PROGRAM PRG_PID_CALL
VAR
	fbPlantControl : PlantAndCMs.FB_PlantControl_mode_2;
	Udt_FbPlantControl : PlantAndCMs.Udt_PlantControl_Mode_2;
	
	fbPlantModeSelector : PlantAndCMs.FB_ModeSelector;
	Udt_PlantModeSelector : PlantAndCMs.Udt_ModeSelector;
END_VAR

//aiSpare02c AT %I*: INT; //ch3 0-10v  Legacy range			(0-32767)
//measure 0-10v
//GVL.rAIInput1 := (INT_TO_REAL(IO.aiSpare02c)/(32767.0-0.0)) * 10.0;

//aiSpare02d AT %I*: INT; //ch4 0-20mA Extended range 		(0 -30518)
//measure 0-100%
//GVL.rAIInput2 := (INT_TO_REAL(IO.aiSpare02d)/(30518.0-0.0)) * 100.0;
fbPlantModeSelector(
	Ctrl_Data_ModeSelector := Udt_PlantModeSelector
	);

	
fbPlantControl(
	Start_In := PlantAndCMs.FIO.bStart,
	Stop_In := PlantAndCMs.FIO.bStop, 
	Reset_In := PlantAndCMs.FIO.bReset,
	
	
	Ctrl_Plant := Udt_FbPlantControl
	);

IF fbPlantControl.Startet_Out THEN
	//PRG_FB_CTRL_PID.bInit := TRUE;
	PRG_FB_CTRL_PID(
	
	);
END_IF

END_PROGRAM

(* stored: Version 1.1.0.1, ProductVersion 3.1.4024.13
   POU PRG_PID_CALL: Id {e7fc84ae-b95c-477c-b1bf-9630c0dddc70}, SpecialFunc None *)
